FUNCTION func_f1: BOOL
VAR_INPUT
    farg_f1_p: BOOL;
END_VAR

func_f1 := (farg_f1_p) AND (ifExprFunc1(dummy:=0));
RETURN;

END_FUNCTION

(* stored: ProductVersion 3.1.0.18, Version 1.1.0.1 *)
